FUNCTION_BLOCK CanisterCounter
  (* Standard: 61499-2 *)
  (* Version 0.1, 2016-00-28, hpea485, UOA *)
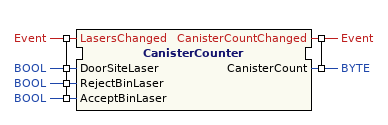
  EVENT_INPUT
    LasersChanged WITH DoorSiteLaser, RejectBinLaser, AcceptBinLaser;
  END_EVENT
  EVENT_OUTPUT
    CanisterCountChanged WITH CanisterCount;
  END_EVENT
  VAR_INPUT
    DoorSiteLaser : BOOL;
    RejectBinLaser : BOOL;
    AcceptBinLaser : BOOL;
  END_VAR
  VAR_OUTPUT
    CanisterCount : BYTE;
  END_VAR
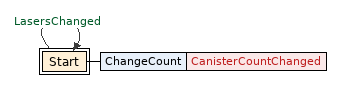
  EC_STATES
    Start : ChangeCount -> CanisterCountChanged;
  END_STATES
  EC_TRANSITIONS
    Start TO Start := LasersChanged;
  END_TRANSITIONS
  ALGORITHM ChangeCount IN ST:
if DoorSiteLaser then
	CanisterCount := CanisterCount + 1;
end_if;
if RejectBinLaser then
	CanisterCount := CanisterCount - 1;
end_if;
if AcceptBinLaser then
	CanisterCount := CanisterCount - 1;
end_if;
  END_ALGORITHM
END_FUNCTION_BLOCK
